FUNCTION_BLOCK PS_PackML_UnitModeManager
VAR_INPUT
	bExecute						:				BOOL;
	ePMLUnitModeCommand				:				E_PMLUnitMode;
	ePMLState						:				E_PMLState;
END_VAR
VAR_OUTPUT
	ePMLUnitModeStatus				:				E_PMLUnitMode;
	bDone							:				BOOL;
	bError							:				BOOL;
	nErrorID						:				UDINT;
END_VAR
VAR
	fbTriggerModeChange					:				R_TRIG;
END_VAR


	fbTriggerModeChange(CLK	:=	bExecute);

	IF fbTriggerModeChange.Q THEN
		bDone			:=		FALSE;
		bError			:=		FALSE;
		nErrorID		:=		0;
		
		CASE ePMLUnitModeStatus OF
			
			E_PMLUnitMode.UNDEFINED:
					ePMLUnitModeStatus	:=	ePMLUnitModeCommand;
					bDone				:=	TRUE;
			
			E_PMLUnitMode.AUTOMATIC:
					IF (ePMLState = E_PMLState.ABORTED) OR (ePMLState = E_PMLState.STOPPED) OR (ePMLState = E_PMLState.IDLE) THEN
						ePMLUnitModeStatus	:=	ePMLUnitModeCommand;
						bDone				:=	TRUE;
					ELSIF ((ePMLState = E_PMLState.HELD) OR (ePMLState = E_PMLState.SUSPENDED) OR (ePMLState = E_PMLState.COMPLETE))
						AND (ePMLUnitModeCommand = E_PMLUnitMode.SEMIAUTOMATIC) THEN
							ePMLUnitModeStatus	:=	ePMLUnitModeCommand;
							bDone				:=	TRUE;
					ELSIF (ePMLState = E_PMLState.HELD) AND (ePMLUnitModeCommand = E_PMLUnitMode.MAINTENANCE) THEN
							ePMLUnitModeStatus	:=	ePMLUnitModeCommand;
							bDone				:=	TRUE;
					ELSE
							bDone				:=	FALSE;
							bError				:=	TRUE;
							nErrorID			:=	1;
					END_IF
			E_PMLUnitMode.SEMIAUTOMATIC:
					IF (ePMLState = E_PMLState.ABORTED) OR (ePMLState = E_PMLState.STOPPED) OR (ePMLState = E_PMLState.IDLE) THEN
						ePMLUnitModeStatus	:=	ePMLUnitModeCommand;
						bDone				:=	TRUE;
					ELSIF ((ePMLState = E_PMLState.HELD) OR (ePMLState = E_PMLState.SUSPENDED) OR (ePMLState = E_PMLState.COMPLETE))
						AND (ePMLUnitModeCommand = E_PMLUnitMode.AUTOMATIC) THEN
							ePMLUnitModeStatus	:=	ePMLUnitModeCommand;
							bDone				:=	TRUE;
					ELSIF (ePMLState = E_PMLState.HELD) AND (ePMLUnitModeCommand = E_PMLUnitMode.MAINTENANCE) THEN
							ePMLUnitModeStatus	:=	ePMLUnitModeCommand;
							bDone				:=	TRUE;
					ELSE
							bDone				:=	FALSE;
							bError				:=	TRUE;
							nErrorID			:=	1;
					END_IF
			E_PMLUnitMode.MANUAL:
					IF (ePMLState = E_PMLState.ABORTED) OR (ePMLState = E_PMLState.STOPPED) OR (ePMLState = E_PMLState.IDLE) THEN
						ePMLUnitModeStatus	:=	ePMLUnitModeCommand;
						bDone				:=	TRUE;
					ELSE
							bDone				:=	FALSE;
							bError				:=	TRUE;
							nErrorID			:=	1;
					END_IF					
			E_PMLUnitMode.MAINTENANCE:
					IF (ePMLState = E_PMLState.ABORTED) OR (ePMLState = E_PMLState.STOPPED) OR (ePMLState = E_PMLState.IDLE) THEN
						ePMLUnitModeStatus	:=	ePMLUnitModeCommand;
						bDone				:=	TRUE;
					ELSIF (ePMLState = E_PMLState.HELD) AND ((ePMLUnitModeCommand = E_PMLUnitMode.AUTOMATIC) OR (ePMLUnitModeCommand = E_PMLUnitMode.SEMIAUTOMATIC)) THEN
							ePMLUnitModeStatus	:=	ePMLUnitModeCommand;
							bDone				:=	TRUE;
					ELSE
							bDone				:=	FALSE;
							bError				:=	TRUE;
							nErrorID			:=	1;
					END_IF					
					
			E_PMLUnitMode.DRYRUN:
					ePMLUnitModeStatus	:=	ePMLUnitModeCommand;
					bDone				:=	TRUE;
					
			E_PMLUnitMode.USERMODE1:
					ePMLUnitModeStatus	:=	ePMLUnitModeCommand;
					bDone				:=	TRUE;
					
			E_PMLUnitMode.USERMODE2:
					ePMLUnitModeStatus	:=	ePMLUnitModeCommand;
					bDone				:=	TRUE;
					
			E_PMLUnitMode.IDLE:
					IF (ePMLState = E_PMLState.ABORTED) OR (ePMLState = E_PMLState.STOPPED) OR (ePMLState = E_PMLState.IDLE) THEN
						ePMLUnitModeStatus	:=	ePMLUnitModeCommand;
						bDone				:=	TRUE;
					ELSE
							bDone				:=	FALSE;
							bError				:=	TRUE;
							nErrorID			:=	1;
					END_IF
			E_PMLUnitMode.ESTOP:
					IF (ePMLState = E_PMLState.ABORTED) OR (ePMLState = E_PMLState.STOPPED) OR (ePMLState = E_PMLState.IDLE) THEN
						ePMLUnitModeStatus	:=	ePMLUnitModeCommand;
						bDone				:=	TRUE;
					ELSE
							bDone				:=	FALSE;
							bError				:=	TRUE;
							nErrorID			:=	1;
					END_IF
		END_CASE
	END_IF

END_FUNCTION_BLOCK

(* stored: Version 1.1.0.1, ProductVersion 3.1.4024.15
   POU PS_PackML_UnitModeManager: Id {dc4f20d7-6b30-44fa-9729-9733db7a4e11}, SpecialFunc None *)
